FUNCTION_BLOCK Place_Services (* Basic Function Block Type *)
  (* Standard: 61499-2 *)
  (* Version 0.0, 11/3/2020, prana, nxtControl GmbH, Template *)
  PACKAGE Main;
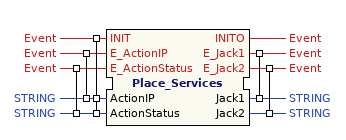
  EVENT_INPUT
    INIT WITH ActionIP, ActionStatus; (* Initialization Request *)
    E_ActionIP WITH ActionIP; (* Normal Execution Request *)
    E_ActionStatus WITH ActionStatus;
  END_EVENT
  EVENT_OUTPUT
    INITO; (* Initialization Confirm *)
    E_Jack1 WITH Jack1;
    E_Jack2 WITH Jack2;
  END_EVENT
  VAR_INPUT
    ActionIP : STRING; (* Input event qualifier *)
    ActionStatus : STRING;
  END_VAR
  VAR_OUTPUT
    Jack1 : STRING;
    Jack2 : STRING;
  END_VAR
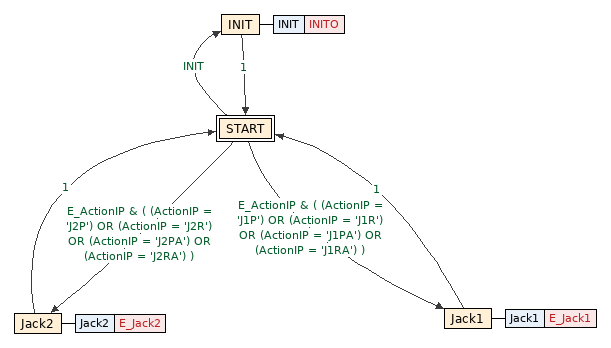
  EC_STATES
    START; (* Initial State *)
    INIT : INIT -> INITO; (* Initialization *)
    Jack1 : Jack1 -> E_Jack1;
    Jack2 : Jack2 -> E_Jack2;
  END_STATES
  EC_TRANSITIONS
    START TO INIT := INIT;
    INIT TO START := 1;
    START TO Jack1 := E_ActionIP & ( (ActionIP = 'J1P') OR (ActionIP = 'J1R') OR (ActionIP = 'J1PA') OR (ActionIP = 'J1RA') );
    Jack1 TO START := 1;
    START TO Jack2 := E_ActionIP & ( (ActionIP = 'J2P') OR (ActionIP = 'J2R') OR (ActionIP = 'J2PA') OR (ActionIP = 'J2RA') );
    Jack2 TO START := 1;
  END_TRANSITIONS
  ALGORITHM INIT IN ST: (* Initialization algorithm *)
;
  END_ALGORITHM
  ALGORITHM REQ IN ST: (* Normally executed algorithm *)
;
  END_ALGORITHM
  ALGORITHM Jack1 IN ST:
Jack1 := ActionIP;
  END_ALGORITHM
  ALGORITHM Jack2 IN ST:
Jack2 := ActionIP;
  END_ALGORITHM
END_FUNCTION_BLOCK
